RoboDK station: Funciona(3).rdk

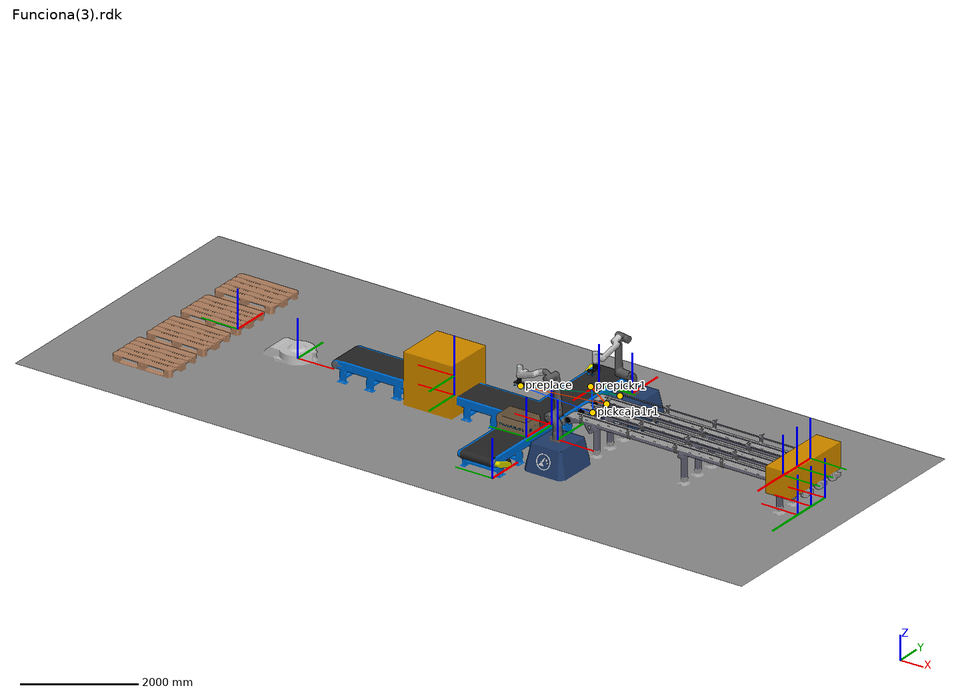
[picture v0: the station drawn from its stored meshes, robots at their saved joint values, targets as dots, program paths as lines]
Station Funciona(3) (saved by RoboDK 5.7.4). Poses are relative to the parent item; angles as X-Y-Z fixed-axis rotations.
  - folder Cintas Pequenyas
    - frame cinta1 at (4400, 800, 0) mm, rotated rx 0 ry 0 rz 180 deg
      - robot cinta1c: 1 axes
          modified DH rows (alpha deg, a mm, theta deg, d mm): 0, 0, 0, 0 linear
          base shift (0, 0, 0) mm, rotated rx 0 ry 90 rz 0 deg
          joint limits [-900000] to [900000]; home [0]; saved at [0]
        - frame caja1f at (300, 0, 0) mm, rotated rx 0 ry 0 rz 90 deg
          - object caja1 at (0, 0, 0) mm, size 199 x 305.1 x 133.7 mm, geometry from Box-12x7in-Closed.sld
      - target inicinta1 (joint target) at (0, 0, 663) mm; joints [0, 0, 0, 0, 0, 0] of cinta1c
      - target fincinta1 (joint target) at (4000, 0, 663) mm; joints [4000, 0, 0, 0, 0, 0] of cinta1c
      - object spawn1 at (-150, -50, 500) mm, size 500 x 500 x 500 mm, geometry from Cube-500mm.sld
    - frame cinta2 at (4400, 1200, 0) mm, rotated rx 0 ry 0 rz 180 deg
      - robot cinta2c: 1 axes
          modified DH rows (alpha deg, a mm, theta deg, d mm): 0, 0, 0, 0 linear
          base shift (0, 0, 0) mm, rotated rx 0 ry 90 rz 0 deg
          joint limits [-900000] to [900000]; home [0]; saved at [0]
        - frame caja2f at (300, 0, 0) mm, rotated rx 0 ry 0 rz 90 deg
          - object caja2 at (0, 0, 0) mm, size 199 x 305.1 x 133.7 mm, geometry from Box-12x7in-Closed.sld
      - target inicinta2 (joint target) at (0, 0, 663) mm; joints [0, 6.328, -12.115, 76.186, 22.998, -75.045] of cinta2c
      - target fincinta2 (joint target) at (4000, 0, 663) mm; joints [4000, 6.328, -12.115, 76.186, 22.998, -75.045] of cinta2c
      - object spawn2 at (-150, -150, 500) mm, size 500 x 500 x 500 mm, geometry from Cube-500mm.sld
    - frame cinta3 at (4400, 1600, 0) mm, rotated rx 0 ry 0 rz 180 deg
      - robot cinta3c: 1 axes
          modified DH rows (alpha deg, a mm, theta deg, d mm): 0, 0, 0, 0 linear
          base shift (0, 0, 0) mm, rotated rx 0 ry 90 rz 0 deg
          joint limits [-900000] to [900000]; home [0]; saved at [0]
        - frame caja3f at (300, 0, 0) mm, rotated rx 0 ry 0 rz 90 deg
          - object caja3 at (0, 0, 0) mm, size 199 x 305.1 x 133.7 mm, geometry from Box-12x7in-Closed.sld
      - target inicinta3 (joint target) at (0, 0, 663) mm; joints [0, 26.9, -39.102, 77.057, 43.994, -72.284] of cinta3c
      - target fincinta3 (joint target) at (4000, 0, 663) mm; joints [4000, 26.9, -39.102, 77.057, 43.994, -72.284] of cinta3c
      - object spawn3 at (-150, -250, 500) mm, size 500 x 500 x 500 mm, geometry from Cube-500mm.sld
  - folder Cintas Grandes
    - frame cintag1 at (-650, -1000, 0) mm, rotated rx 0 ry 0 rz 90 deg
      - robot cintag1c: 1 axes
          modified DH rows (alpha deg, a mm, theta deg, d mm): 0, 0, 0, 0 linear
          base shift (0, 0, 0) mm, rotated rx 0 ry 90 rz 0 deg
          joint limits [-900000] to [900000]; home [0]; saved at [1000]
        - frame cajag1f at (0, 0, 0) mm
          - object cajag1 at (0, 0, 0) mm, size 424.8 x 637.2 x 266.3 mm, geometry from Box-24x16in-Open.sld
      - target inicintag1 (joint target) at (0, 0, 366.5) mm; joints [0, -12.476, 26.215, 0, 76.261, 75.584] of cintag1c
      - target medcintag1 (joint target) at (1000, 0, 366.5) mm; joints [1000, -12.476, 26.215, 0, 76.261, 75.584] of cintag1c
      - target fincintag1 (joint target) at (1500, 0, 366.5) mm; joints [1500, -12.476, 26.215, 0, 76.261, 75.584] of cintag1c
    - frame cintag2 at (-1250, 3000, 0) mm, rotated rx 0 ry 0 rz -90 deg
      - robot cintag2c: 1 axes
          modified DH rows (alpha deg, a mm, theta deg, d mm): 0, 0, 0, 0 linear
          base shift (0, 0, 0) mm, rotated rx 0 ry 90 rz 0 deg
          joint limits [-900000] to [900000]; home [0]; saved at [0]
    - frame cintag3 at (-1000, 1250, 0) mm, rotated rx 0 ry 0 rz 180 deg
      - robot cintag3c: 1 axes
          modified DH rows (alpha deg, a mm, theta deg, d mm): 0, 0, 0, 0 linear
          base shift (0, 0, 0) mm, rotated rx 0 ry 90 rz 0 deg
          joint limits [-900000] to [900000]; home [0]; saved at [0]
    - frame cintag4 at (-3000, 1250, 0) mm, rotated rx 0 ry 0 rz 180 deg
      - robot cintag4c: 1 axes
          modified DH rows (alpha deg, a mm, theta deg, d mm): 0, 0, 0, 0 linear
          base shift (0, 0, 0) mm, rotated rx 0 ry 90 rz 0 deg
          joint limits [-900000] to [900000]; home [0]; saved at [0]
        - frame cajag3f at (0, 0, 0) mm
          - object cajag3 at (0, 0, 0) mm, size 424.8 x 637.2 x 266.3 mm, geometry from Box-24x16in-Open.sld
      - object precint at (-500, -200, 0) mm, size 1000 x 1000 x 1000 mm, geometry from Cube-1000mm.sld
  - folder Pisos
    - object Floor at (700, -500, 0) mm, size 3000 x 3000 x 0 mm, geometry from Floor.sld
    - object Floor1 at (3700, -500, 0) mm, size 3000 x 3000 x 0 mm, geometry from Floor.sld
    - object Floor2 at (-2300, -500, 0) mm, size 3000 x 3000 x 0 mm, geometry from Floor.sld
    - object Floor3 at (3700, 2500, 0) mm, size 3000 x 3000 x 0 mm, geometry from Floor.sld
    - object Floor4 at (700, 2500, 0) mm, size 3000 x 3000 x 0 mm, geometry from Floor.sld
    - object Floor5 at (-2300, 2500, 0) mm, size 3000 x 3000 x 0 mm, geometry from Floor.sld
    - object Floor6 at (-5300, -500, 0) mm, size 3000 x 3000 x 0 mm, geometry from Floor.sld
    - object Floor7 at (-5300, 2500, 0) mm, size 3000 x 3000 x 0 mm, geometry from Floor.sld
    - object Floor8 at (-8300, 2500, 0) mm, size 3000 x 3000 x 0 mm, geometry from Floor.sld
    - object Floor9 at (-8300, -500, 0) mm, size 3000 x 3000 x 0 mm, geometry from Floor.sld
  - folder Robots P&P
    - object pedestal at (0, 0, 0) mm, size 844.5 x 933.7 x 500 mm, geometry from Pedestal-H500mm-Type-2.sld
    - frame robot1 at (0, 0, 500) mm
      - robot robot1c (model ABB CRB 15000 10): 6 axes
          modified DH rows (alpha deg, a mm, theta deg, d mm): 0, 0, 0, 400; -90, 150, -90, 0; 0, 707, 0, 0; -90, 110, 0, 637; 90, 0, 0, 0; -90, 80, 180, 101
          joint limits [-270, -180, -225, -180, -180, -270] to [270, 180, 85, 180, 180, 270]; home [0, 0, 0, 0, 0, 0]; saved at [170.764, 2.845, 18.663, 0, 68.493, 170.764]
        - tool vacuum1, TCP at (0, 30, 180) mm, size 239 x 147 x 184.9 mm
      - target prepickr1 (Cartesian target) at (179.79, 729.43, 764.88) mm, rotated rx 180 ry 0 rz -180 deg; joints [75.584, -12.476, 26.215, 0, 76.261, 75.584] of robot1c
      - target pickcaja1r1 (Cartesian target) at (242.56, 692.28, 298.87) mm, rotated rx -180 ry 0 rz 180 deg; joints [69.885, 7.532, 55.973, 0, 26.494, 69.885] of robot1c
      - target pickcaja2r1 (Cartesian target) at (242.56, 1100, 298.87) mm, rotated rx -180 ry 0 rz -180 deg; joints [77.227, 32.053, 18.191, 0, 39.757, 77.227] of robot1c
      - target pickcaja3r1 (Cartesian target) at (242.56, 1500, 298.87) mm, rotated rx -180 ry 0 rz 180 deg; joints [80.63, 62.888, -40.371, 0, 67.483, 80.63] of robot1c
      - target preplace (Cartesian target) at (-886.42, 174.14, 693.93) mm, rotated rx -180 ry 0 rz 180 deg; joints [170.764, 2.845, 18.663, 0, 68.493, 170.764] of robot1c
      - target place1 (Cartesian target) at (-886.42, 174.14, 693.93) mm, rotated rx -180 ry 0 rz 180 deg; joints [170.764, 2.845, 18.663, 0, 68.493, 170.764] of robot1c
    - object pedestal2 at (0, 2200, 0) mm, size 844.5 x 933.7 x 500 mm, geometry from Pedestal-H500mm-Type-2.sld
    - frame robot2 at (0, 2200, 500) mm, rotated rx 0 ry 0 rz 90 deg
      - robot robot2c (model ABB CRB 15000 10): 6 axes
          modified DH rows (alpha deg, a mm, theta deg, d mm): 0, 0, 0, 400; -90, 150, -90, 0; 0, 707, 0, 0; -90, 110, 0, 637; 90, 0, 0, 0; -90, 80, 180, 101
          joint limits [-270, -180, -225, -180, -180, -270] to [270, 180, 85, 180, 180, 270]; home [0, 0, 0, 0, 0, 0]; saved at [170.764, 2.845, 18.663, 0, 68.493, 170.764]
        - tool vacuum2, TCP at (0, 30, 180) mm, size 239 x 147 x 184.9 mm
  - folder Robot Pallet
    - frame robot3 at (-6000, 900, 0) mm
      - robot robot3c (model ABB IRB 4400/L30 M2000): 6 axes, payload 30 kg, reach 2432 mm, repeatability 0.2 mm, weight 1040 kg
          joint limits [-165, -70, -165, -200, -120, -400] to [165, 95, 165, 200, 120, 400]; home [0, 0, 0, 0, 0, 0]; saved at [0, 0, 0, 0, 0, 0]
        - tool vacuum3, TCP at (-36, 0, 106.49) mm, size 268.4 x 184.1 x 103.7 mm
      - frame pallets at (-1300, 100, 150) mm, rotated rx 0 ry 0 rz 90 deg
        - object pallet1 at (1000, 0, 0) mm, size 800 x 1200 x 144.2 mm, geometry from Pallet-1200x800mm-Transverse.sld
        - object pallet2 at (0, 0, 0) mm, size 800 x 1200 x 144.2 mm, geometry from Pallet-1200x800mm-Transverse.sld
        - object pallet3 at (-1000, 0, 0) mm, size 800 x 1200 x 144.2 mm, geometry from Pallet-1200x800mm-Transverse.sld
        - object pallet4 at (-2000, 0, 0) mm, size 800 x 1200 x 144.2 mm, geometry from Pallet-1200x800mm-Transverse.sld
  - folder Pick & Place 1
    - program p&p_caja1 (6 instructions, listed below)
    - program p&p_caja2 (6 instructions, listed below)
    - program p&p_caja3 (6 instructions, listed below)
  - folder MQTT
    - Python program MqttListener (listed below)
    - Python program RobotController (listed below)
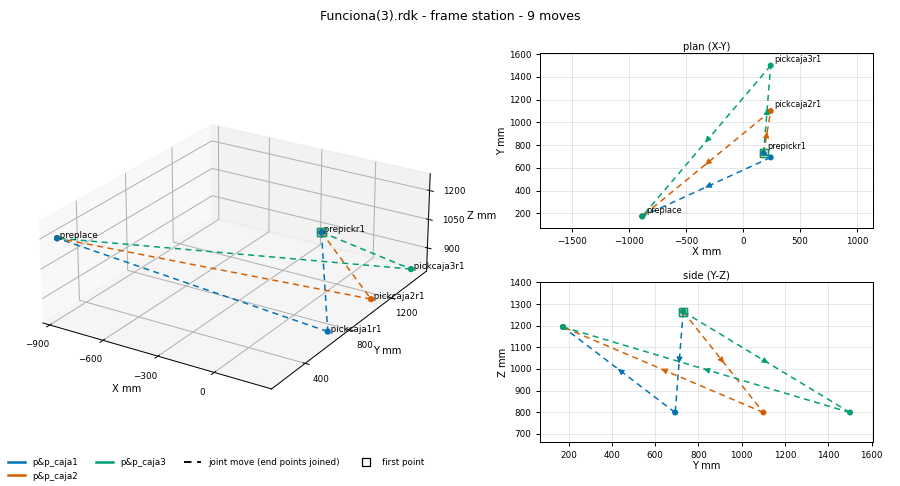
[picture p0: tool path of Funciona(3).rdk in frame station, 9 of 9 moves have a stored position in this frame; points joined in program order, loops and branches not executed]

--- program p&p_caja1 (robot robot1c) ---
  Est. Ref.: robot1
  Est. herr: vacuum1
  MoveJ (prepickr1)
  MoveJ (pickcaja1r1)
  Adjuntar a vacuum1
  MoveJ (preplace)

--- program p&p_caja2 (robot robot1c) ---
  Est. Ref.: robot1
  Est. herr: vacuum1
  MoveJ (prepickr1)
  MoveJ (pickcaja2r1)
  Adjuntar a vacuum1
  MoveJ (preplace)

--- program p&p_caja3 (robot robot1c) ---
  Est. Ref.: robot1
  Est. herr: vacuum1
  MoveJ (prepickr1)
  MoveJ (pickcaja3r1)
  Adjuntar a vacuum1
  MoveJ (preplace)

--- Python program MqttListener ---
from robodk import robolink
RDK = robolink.Robolink()

import paho.mqtt.client as mqtt
import RobotController as rc

broker = "mqtt.dsic.upv.es"
port = 1883
user = "giirob"
passwd = "UPV2024"

topic_sub = "giirob/pr2/station/demo/commands"
topic_pub = "giirob/pr2/station/demo/status"


def on_message(mqttc, obj, msg):
    payload = msg.payload.decode('utf-8')
    topic = msg.topic
    qos = msg.qos
    rc.handle_message(mqttc, topic, payload)

mqttc = mqtt.Client(mqtt.CallbackAPIVersion.VERSION2)
mqttc.on_message = on_message

mqttc.username_pw_set(username=user, password=passwd)
mqttc.connect(broker, port, 60)
mqttc.subscribe(topic_sub, 0)

mqttc.publish(topic_pub, "ready 1")


mqttc.loop_forever()

--- Python program RobotController ---
from robodk import robolink
from robodk.robolink import ITEM_TYPE_PROGRAM
import threading

RDK = robolink.Robolink()

import paho.mqtt.client as mqtt

station_commands_topic = "giirob/pr2/station/demo/commands"
station_status_topic = "giirob/pr2/station/demo/status"


def handle_message(mqttc, topic, payload):
    msg = payload.strip()

    print(" Mensaje recibido:", msg)

    if topic == station_commands_topic:


        if msg == "1":
            hilo = threading.Thread(
                target=ejecutar_programa,
                args=(mqttc, "p&p_caja1")
            )
            hilo.start()

        elif msg == "2":
            hilo = threading.Thread(
                target=ejecutar_programa,
                args=(mqttc, "p&p_caja2")
            )
            hilo.start()

         # else:
            #print("Comando no reconocido")


def ejecutar_programa(mqttc, nombre_programa):
    programa = RDK.Item(nombre_programa, ITEM_TYPE_PROGRAM)
    programa.RunProgram()
